FUNCTION FC_SetPartProgramNameByID : STRING
VAR_INPUT
	Id : LINT;
END_VAR
VAR
	sId : STRING;
	str : STRING(9) := 'O00000000';
END_VAR


sId := LINT_TO_STRING(id);
FC_SetPartProgramNameByID := CONCAT(LEFT(str, 9 - LEN(sId)), sId);

END_FUNCTION

(* stored: Version 1.1.0.1, ProductVersion 3.1.4024.13
   POU FC_SetPartProgramNameByID: Id {ce5cdbcc-714c-4d35-b371-1ec2167f2002}, SpecialFunc None *)
